PROGRAM MAIN
VAR
END_VAR

END_PROGRAM

(* stored: Version 1.1.0.1
   POU MAIN: Id {a338f754-6b78-4d00-bd73-d9b8927526a8} *)
